{attribute 'GeneratedUsingTerminal: EP5101-2011-0016'}
{attribute addProperty BoxType "EP5101-2011-0016"}
{attribute addProperty Id "ENC_Status_compactAT %I*ENC_Status_compact_4198EF3B17ENC_Control_compactAT %Q*ENC_Control_compact_21E2D14D6WcStateAT %I*WcState_9091E0EB2InfoDataAT %I*InfoData_32EB74EA10"}
{attribute addProperty CRC "942314159"}
{attribute addProperty Size "35"}
TYPE EP5101_382A92AF EXTENDS EtcSlaveTerminalBase_947E5A46 :
STRUCT
	{attribute addProperty Name "ENC_Status_compact"}
	ENC_Status_compact : ENC_Status_compact_4198EF3B;
	{attribute addProperty Name "ENC_Control_compact"}
	ENC_Control_compact : ENC_Control_compact_21E2D14D;
	{attribute addProperty Name "WcState"}
	WcState : WcState_9091E0EB;
	{attribute addProperty Name "InfoData"}
	InfoData : InfoData_32EB74EA;
END_STRUCT
END_TYPE

(* stored: Version 1.2.0.0, ProductVersion 3.1.4024.9
   DUT EP5101_382A92AF: Id {ccef961f-c25f-4552-9419-10440d7d4009} *)
